// TIA Portal V18 export
TYPE "ST_Conveyer_Line"
// stored: IsFailsafeCompliant false
   STRUCT
      HMI_StartPB : Bool;
      HMI_StopPB : Bool;
      Auto_Start : Bool;
      Auto_Stop : Bool;
      Run : Bool;
      OverLoad : Bool;
   END_STRUCT;
END_TYPE
